// TIA Portal V17 export
// export: Created 2025-06-26T06:49:30.6164939Z, ExportSetting WithDefaults, DisplayName Totally Integrated Automation Portal, DisplayVersion V17 Update 8, DisplayName TIA Portal Openness, DisplayVersion V17 Update 8, DisplayName TIA Portal Version Control Interface, DisplayVersion V17, DisplayName STEP 7 Professional, DisplayVersion V17 Update 8, DisplayName STEP 7 Safety, DisplayVersion V17 Update 6, DisplayName WinCC Advanced, DisplayVersion V17 Update 8
TYPE "stTemperatureController2"
// stored: IsFailsafeCompliant false
   STRUCT
      bEnable : Bool;   // 1 = controller active, 0 = controller inactive
      fHeatingSetpoint : Real;   // When below this temp, begin heating
      fCoolingSetpoint : Real;   // When above this temp, begin cooling
      bHeating : Bool;   // 1 = heating on, 0 = heating off
      bCooling : Bool;   // 1 = cooling on, 0 = cooling off
      bAtSetpoint : Bool;   // 1 = at setpoint, 0 = not at setpoint
      bFault : Bool;   // 1 = controller fault, 0 = ok
      bManualMode : Bool;   // 1 = manual setpoint, 0 = normal
      fManualHeatingSetpoint : Real;
      fManualCoolingSetpoint : Real;
      bManualOverride : Bool;   // 1 = enable forcing outputs
      nOverrideState : USInt;   // 0 = off, 1 = heating, 2 = cooling
      nMode : USInt;   // 0 = Off, 1 = Auto, 2 = Manual, 3 = Manual Override
   END_STRUCT;
END_TYPE
